FUNCTION_BLOCK ServoECAT
VAR_IN_OUT CONSTANT
	bEnable : BOOL;
END_VAR
VAR_OUTPUT
	home AT %I* : BOOL;
	outerLimit AT %I* : BOOL;
	innerLimit AT %I* : BOOL;
	
	ready : BOOL;
	busy : BOOL;
	error : BOOL;
	homeSet : BOOL;
END_VAR
VAR
	axis : AXIS_REF;
	
	mcPower : MC_Power;
	mcMoveAbsolute : MC_MoveAbsolute;
	mcMoveRelative : MC_MoveRelative;
	mcMoveVelocity : MC_MoveVelocity;
	mcSetPosition : MC_SetPosition;
	mcReset : MC_Reset;
	mcStop : MC_Stop;
	
	step : Homing;
END_VAR
VAR
	
END_VAR

mcReset(
	Axis:= axis, 
	Execute:= , 
	Done=> , 
	Busy=> , 
	Error=> , 
	ErrorID=> );

IF mcReset.Execute AND mcReset.Done THEN
	mcReset.Execute := FALSE;
END_IF

mcPower(
	Axis:= axis, 
	Enable:= bEnable, 
	Enable_Positive:= TRUE, 
	Enable_Negative:= TRUE, 
	Override:= 100, 
	BufferMode:= , 
	Options:= , 
	Status=> , 
	Busy=> , 
	Active=> , 
	Error=> , 
	ErrorID=> );

mcMoveAbsolute(
	Axis:= axis, 
	Execute:= , 
	Position:= , 
	Velocity:= 500, 
	Acceleration:= , 
	Deceleration:= , 
	Jerk:= , 
	BufferMode:= , 
	Options:= , 
	Done=> , 
	Busy=> , 
	Active=> , 
	CommandAborted=> , 
	Error=> , 
	ErrorID=> );
	
mcMoveRelative(
	Axis:= axis, 
	Execute:= , 
	Distance:= ,
	Velocity:= 500, 
	Acceleration:= , 
	Deceleration:= , 
	Jerk:= , 
	BufferMode:= , 
	Options:= , 
	Done=> , 
	Busy=> , 
	Active=> , 
	CommandAborted=> , 
	Error=> , 
	ErrorID=> );
	
mcMoveVelocity(
	Axis:= axis, 
	Execute:= , 
	Velocity:= 200, 
	Acceleration:= , 
	Deceleration:= , 
	Jerk:= , 
	Direction:= , 
	BufferMode:= , 
	Options:= , 
	InVelocity=> , 
	Busy=> , 
	Active=> , 
	CommandAborted=> , 
	Error=> , 
	ErrorID=> );

busy := mcMoveAbsolute.Busy OR mcMoveRelative.Busy OR mcMoveVelocity.Busy OR mcSetPosition.Busy OR mcReset.Busy OR mcStop.Busy OR step <> 0;
error := mcMoveAbsolute.Error OR mcMoveRelative.Error OR mcMoveVelocity.Error OR mcSetPosition.Error OR mcReset.Error OR mcStop.Error OR step <> 0;
	
ready := bEnable AND NOT busy AND homeSet;

METHOD homingSequence : BOOL
CASE step OF
	Homing.IDLE:
		mcStop.Execute := FALSE;
		step := Homing.REDO;
		
	Homing.REDO:
		mcMoveVelocity.Direction := MC_Negative_Direction;
		mcMoveVelocity.Execute := TRUE;
		
		IF NOT innerLimit THEN
			
			mcMoveVelocity.Execute := FALSE;
			step := Homing.HOME_OUT;
		END_IF
		
	Homing.HOME_OUT:
		mcMoveVelocity.Direction := MC_Positive_Direction;
		mcMoveVelocity.Execute := TRUE;
		
		IF NOT homingSequence THEN //if reached home
			mcMoveVelocity.Execute := FALSE;
			step := Homing.STOP;
		END_IF
		
	Homing.STOP:
		mcStop.Execute := TRUE;
		IF mcStop.Done THEN
			mcStop.Execute := FALSE;
			step := Homing.SET;
		END_IF
		
	Homing.SET:
		mcSetPosition.Position := 0;
		mcSetPosition.Execute := TRUE;
		
		IF mcSetPosition.Done THEN
			mcSetPosition.Execute := FALSE;
			step := Homing.IDLE;
		END_IF
		
	
END_CASE
END_METHOD

METHOD moveAbsolute : BOOL
VAR_INPUT
	position : LREAL;
END_VAR
VAR_OUTPUT
	fault : BOOL;
END_VAR
IF NOT busy AND NOT error THEN
	mcMoveAbsolute.Position := position;
END_IF
moveAbsolute := mcMoveAbsolute.Done;
END_METHOD

METHOD moveContinuous : BOOL
VAR_INPUT
	direction : BOOL; //direction (F = inwards, T = outwards)
END_VAR
IF direction THEN
	mcMoveVelocity.Direction := MC_Positive_Direction;
ELSE
	mcMoveVelocity.Direction := MC_Negative_Direction;
END_IF

mcMoveVelocity.Execute := TRUE;
moveContinuous := TRUE;
END_METHOD

METHOD moveRelative : BOOL
VAR_INPUT
	distance : LREAL;
END_VAR
mcMoveRelative.Distance := distance;

moveRelative := mcMoveRelative.Done;
END_METHOD

METHOD reset : BOOL
VAR_INPUT
END_VAR
mcReset.Execute := TRUE;

reset := mcReset.Done;
END_METHOD

METHOD stop : BOOL
VAR_INPUT
END_VAR
END_METHOD

END_FUNCTION_BLOCK

(* stored: Version 1.1.0.1, ProductVersion 3.1.4024.11
   POU ServoECAT: Id {f939ae28-30bd-4997-8b95-af50702e8d64}, SpecialFunc None
   Method homingSequence: Id {c889c79b-08e7-46ba-b03a-e3652fe9a7a9}
   Method moveAbsolute: Id {9a0c1523-e496-48d2-89d9-d71629c86307}
   Method moveContinuous: Id {c1bd97e2-f7e7-45ed-bf81-7afd3b7c53ff}
   Method moveRelative: Id {a4516e41-c115-4d38-aa54-f9462db8dc0d}
   Method reset: Id {b7706fbc-8e49-4562-bc6d-21f87f45b14e}
   Method stop: Id {131a01d5-9f85-446c-9242-ad02c99596c6} *)
